Staubli VAL3: SplitNumS.pgx

public program SplitNumS(string x_Source (dimensions=1), num& x_Res[] (dimensions=1), string& x_sChar[] (dimensions=1), bool& x_bRes (dimensions=1))
  local num l_nNum
begin

  call SplitString(x_Source,sBuff,x_sChar,x_bRes)
  if !x_bRes
    return
  endIf



  //把分解的字符串转化为数字量
  for l_nNum=0 to min(size(sBuff)-1,size(x_Res)-1)
    toNum(sBuff[l_nNum],x_Res[l_nNum],x_bRes)
    if !x_bRes
      return
    endIf
  endFor




end
